// TIA Portal V20 export
DATA_BLOCK "MotionTemp_DB"   // DB314
// stored: InstanceOfName MotionTemp, InstanceOfType FB
"MotionTemp"
   // VAR
   //    mcPower { S7_SetPoint := 'True'} : Array[1..50] of MC_POWER;
   //    mcHome { S7_SetPoint := 'True'} : Array[1..50] of MC_HOME;
   //    statOn { S7_SetPoint := 'True'} : Bool;
   //    instServoOnTriggerr : R_TRIG;
   // END_VAR
BEGIN
END_DATA_BLOCK
